(* Logix 5000 project; controller p65 vendor 1 type 14 code 85 rev 20.11; software revision 20.01; part 4 of 7 *)
(* tags used below, declared in another part *)
   DCMicroGridisInOperation : ALIAS FOR DINT00_23.8;
   DCMicroGridisSimulating : ALIAS FOR DINT00_23.10;
   House02accountBalance : ALIAS FOR REAL00_128;
   House02accountDepositRate : ALIAS FOR REAL00_129;
   House02Bclose : ALIAS FOR Local:3:O.Data.1;
   House02BcloseHILS : ALIAS FOR plc1_local_6[0].1;
   House02BcloseProxy : ALIAS FOR DINT00_28.31;
   House02BintReqClose : ALIAS FOR DINT00_29.0;
   House02BisClosed : ALIAS FOR DINT00_29.1;
   House02BisOpen : ALIAS FOR DINT00_29.2;
   House02BreqClose : ALIAS FOR DINT00_29.3;
   House02BreqOpen : ALIAS FOR DINT00_29.4;
   House02commandChanged : ALIAS FOR DINT00_29.5;
   House02commandChangedTimer : ALIAS FOR CLTIMER00_57;
   House02current : ALIAS FOR REAL00_130;
   House02currentHILS : ALIAS FOR plc1_local_2[1];
   House02currentRaw : ALIAS FOR Local:1:I.Ch13Data;
   House02deadband : ALIAS FOR REAL00_131;
   House02depositTimer : ALIAS FOR CLTIMER00_58;
   House02DisconnectPowerEventFail : ALIAS FOR DINT00_29.6;
   House02DisconnectPowerEventSuccess : ALIAS FOR DINT00_29.7;
   House02DisconnectPowerFailTimer : ALIAS FOR CLTIMER00_59;
   House02DisconnectPowerInProcess : ALIAS FOR DINT00_29.8;
   House02DisconnectPowerMsg : ALIAS FOR MESSAGE00_14;
   House02DisconnectPowerSuccessTimer : ALIAS FOR CLTIMER00_60;
   House02failedToConnect : ALIAS FOR DINT00_29.9;
   House02failedToDisconnect : ALIAS FOR DINT00_29.10;
   House02fundsAvailable : ALIAS FOR DINT00_29.11;
   House02incrementToAdd : ALIAS FOR REAL00_132;
   House02incrementToSubtract : ALIAS FOR REAL00_133;
   House02intReqConnect : ALIAS FOR DINT00_29.12;
   House02isConnected : ALIAS FOR DINT00_29.13;
   House02isDisconnected : ALIAS FOR DINT00_29.14;
   House02minBalance : ALIAS FOR REAL00_135;
   House02minBalanceToReconnect : ALIAS FOR REAL00_136;
   House02minTime : ALIAS FOR REAL00_137;
   House02powerRate : ALIAS FOR REAL00_138;
   House02powerRateMax : REAL;
   House02PurchasePowerEventFail : ALIAS FOR DINT00_29.15;
   House02PurchasePowerEventSuccess : ALIAS FOR DINT00_29.16;
   House02PurchasePowerFailTimer : ALIAS FOR CLTIMER00_61;
   House02PurchasePowerInProcess : ALIAS FOR DINT00_29.17;
   House02PurchasePowerMsg : ALIAS FOR MESSAGE00_15;
   House02PurchasePowerSuccessTimer : ALIAS FOR CLTIMER00_62;
   House02reqConnect : ALIAS FOR DINT00_29.18;
   House02reqDisconnect : ALIAS FOR DINT00_29.19;
   House02runningOut : ALIAS FOR DINT00_29.20;
   House02spendingRate : ALIAS FOR REAL00_139;
   House02timeRemaining : ALIAS FOR REAL00_140;
   House02usageTimer : ALIAS FOR CLTIMER00_63;
   House03accountBalance : ALIAS FOR REAL00_141;
   House03accountDepositRate : ALIAS FOR REAL00_142;
   House03Bclose : ALIAS FOR Local:3:O.Data.2;
   House03BcloseHILS : ALIAS FOR plc1_local_6[0].2;
   House03BcloseProxy : ALIAS FOR DINT00_29.21;
   House03BintReqClose : ALIAS FOR DINT00_29.22;
   House03BisClosed : ALIAS FOR DINT00_29.23;
   House03BisOpen : ALIAS FOR DINT00_29.24;
   House03BreqClose : ALIAS FOR DINT00_29.25;
   House03BreqOpen : ALIAS FOR DINT00_29.26;
   House03commandChanged : ALIAS FOR DINT00_29.27;
   House03commandChangedTimer : ALIAS FOR CLTIMER00_64;
   House03current : ALIAS FOR REAL00_143;
   House03currentHILS : ALIAS FOR plc1_local_2[2];
   House03currentRaw : ALIAS FOR Local:1:I.Ch14Data;
   House03deadband : ALIAS FOR REAL00_144;
   House03depositTimer : ALIAS FOR CLTIMER00_65;
   House03DisconnectPowerEventFail : ALIAS FOR DINT00_29.28;
   House03DisconnectPowerEventSuccess : ALIAS FOR DINT00_29.29;
   House03DisconnectPowerFailTimer : ALIAS FOR CLTIMER00_66;
   House03DisconnectPowerInProcess : ALIAS FOR DINT00_29.30;
   House03DisconnectPowerMsg : ALIAS FOR MESSAGE00_16;
   House03DisconnectPowerSuccessTimer : ALIAS FOR CLTIMER00_67;
   House03failedToConnect : ALIAS FOR DINT00_29.31;
   House03failedToDisconnect : ALIAS FOR DINT00_30.0;
   House03fundsAvailable : ALIAS FOR DINT00_30.1;
   House03incrementToAdd : ALIAS FOR REAL00_145;
   House03incrementToSubtract : ALIAS FOR REAL00_146;
   House03intReqConnect : ALIAS FOR DINT00_30.2;
   House03isConnected : ALIAS FOR DINT00_30.3;
   House03isDisconnected : ALIAS FOR DINT00_30.4;
   House03minBalance : ALIAS FOR REAL00_148;
   House03minBalanceToReconnect : ALIAS FOR REAL00_149;
   House03minTime : ALIAS FOR REAL00_150;
   House03powerRate : ALIAS FOR REAL00_151;
   House03powerRateMax : REAL;
   House03PurchasePowerEventFail : ALIAS FOR DINT00_30.5;
   House03PurchasePowerEventSuccess : ALIAS FOR DINT00_30.6;
   House03PurchasePowerFailTimer : ALIAS FOR CLTIMER00_68;
   House03PurchasePowerInProcess : ALIAS FOR DINT00_30.7;
   House03PurchasePowerMsg : ALIAS FOR MESSAGE00_17;
   House03PurchasePowerSuccessTimer : ALIAS FOR CLTIMER00_69;
   House03reqConnect : ALIAS FOR DINT00_30.8;
   House03reqDisconnect : ALIAS FOR DINT00_30.9;
   House03runningOut : ALIAS FOR DINT00_30.10;
   House03spendingRate : ALIAS FOR REAL00_152;
   House03timeRemaining : ALIAS FOR REAL00_153;
   House03usageTimer : ALIAS FOR CLTIMER00_70;
   House04accountBalance : ALIAS FOR REAL00_154;
   House04accountDepositRate : ALIAS FOR REAL00_155;
   House04Bclose : ALIAS FOR Local:3:O.Data.3;
   House04BcloseHILS : ALIAS FOR plc1_local_6[0].3;
   House04BcloseProxy : ALIAS FOR DINT00_30.11;
   House04BintReqClose : ALIAS FOR DINT00_30.12;
   House04BisClosed : ALIAS FOR DINT00_30.13;
   House04BisOpen : ALIAS FOR DINT00_30.14;
   House04BreqClose : ALIAS FOR DINT00_30.15;
   House04BreqOpen : ALIAS FOR DINT00_30.16;
   House04commandChanged : ALIAS FOR DINT00_30.17;
   House04commandChangedTimer : ALIAS FOR CLTIMER00_71;
   House04current : ALIAS FOR REAL00_156;
   House04currentHILS : ALIAS FOR plc1_local_2[3];
   House04currentRaw : ALIAS FOR Local:1:I.Ch15Data;
   House04deadband : ALIAS FOR REAL00_157;
   House04depositTimer : ALIAS FOR CLTIMER00_72;
   House04DisconnectPowerEventFail : ALIAS FOR DINT00_30.18;
   House04DisconnectPowerEventSuccess : ALIAS FOR DINT00_30.19;
   House04DisconnectPowerFailTimer : ALIAS FOR CLTIMER00_73;
   House04DisconnectPowerInProcess : ALIAS FOR DINT00_30.20;
   House04DisconnectPowerMsg : ALIAS FOR MESSAGE00_18;
   House04DisconnectPowerSuccessTimer : ALIAS FOR CLTIMER00_74;
   House04failedToConnect : ALIAS FOR DINT00_30.21;
   House04failedToDisconnect : ALIAS FOR DINT00_30.22;
   House04fundsAvailable : ALIAS FOR DINT00_30.23;
   House04incrementToAdd : ALIAS FOR REAL00_158;
   House04incrementToSubtract : ALIAS FOR REAL00_159;
   House04intReqConnect : ALIAS FOR DINT00_30.24;
   House04isConnected : ALIAS FOR DINT00_30.25;
   House04isDisconnected : ALIAS FOR DINT00_30.26;
   House04minBalance : ALIAS FOR REAL00_161;
   House04minBalanceToReconnect : ALIAS FOR REAL00_162;
   House04minTime : ALIAS FOR REAL00_163;
   House04powerRate : ALIAS FOR REAL00_164;
   House04powerRateMax : REAL;
   House04PurchasePowerEventFail : ALIAS FOR DINT00_30.27;
   House04PurchasePowerEventSuccess : ALIAS FOR DINT00_30.28;
   House04PurchasePowerFailTimer : ALIAS FOR CLTIMER00_75;
   House04PurchasePowerInProcess : ALIAS FOR DINT00_30.29;
   House04PurchasePowerMsg : ALIAS FOR MESSAGE00_19;
   House04PurchasePowerSuccessTimer : ALIAS FOR CLTIMER00_76;
   House04reqConnect : ALIAS FOR DINT00_30.30;
   House04reqDisconnect : ALIAS FOR DINT00_30.31;
   House04runningOut : ALIAS FOR DINT00_31.0;
   House04spendingRate : ALIAS FOR REAL00_165;
   House04timeRemaining : ALIAS FOR REAL00_166;
   House04usageTimer : ALIAS FOR CLTIMER00_77;
   LoadslowVoltage : ALIAS FOR DINT00_27.23;
   UsingAgents : BOOL;

PROGRAM House02   (* main routine House02 *)

ROUTINE House02   (* ladder *)
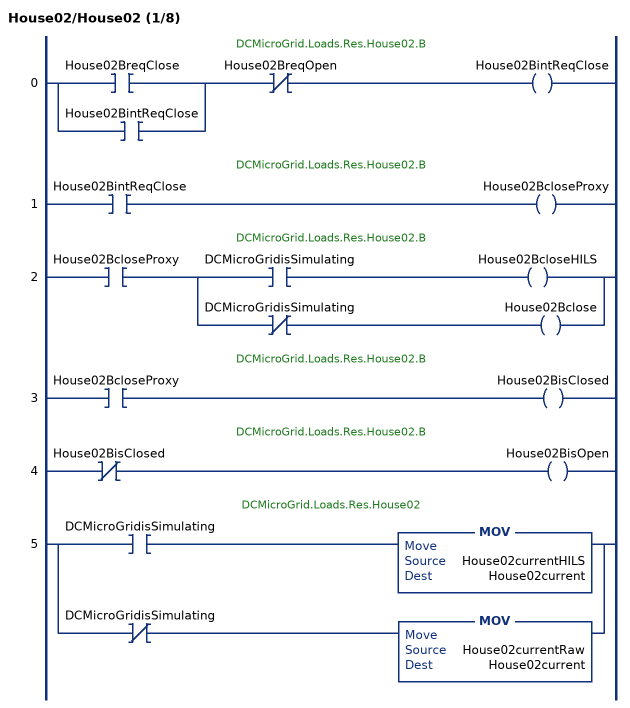
   // DCMicroGrid.Loads.Res.House02.B
   0: [XIC(House02BreqClose) ,XIC(House02BintReqClose) ]XIO(House02BreqOpen)OTE(House02BintReqClose);
   // DCMicroGrid.Loads.Res.House02.B
   1: XIC(House02BintReqClose)OTE(House02BcloseProxy);
   // DCMicroGrid.Loads.Res.House02.B
   2: XIC(House02BcloseProxy)[XIC(DCMicroGridisSimulating) OTE(House02BcloseHILS) ,XIO(DCMicroGridisSimulating) OTE(House02Bclose) ];
   // DCMicroGrid.Loads.Res.House02.B
   3: XIC(House02BcloseProxy)OTE(House02BisClosed);
   // DCMicroGrid.Loads.Res.House02.B
   4: XIO(House02BisClosed)OTE(House02BisOpen);
   // DCMicroGrid.Loads.Res.House02
   5: [XIC(DCMicroGridisSimulating) MOV(House02currentHILS,House02current) ,XIO(DCMicroGridisSimulating) MOV(House02currentRaw,House02current) ];
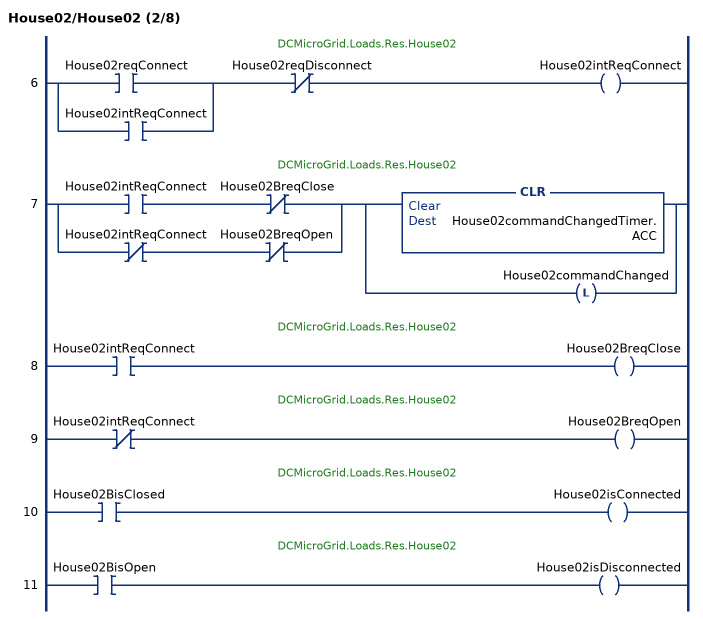
   // DCMicroGrid.Loads.Res.House02
   6: [XIC(House02reqConnect) ,XIC(House02intReqConnect) ]XIO(House02reqDisconnect)OTE(House02intReqConnect);
   // DCMicroGrid.Loads.Res.House02
   7: [XIC(House02intReqConnect) XIO(House02BreqClose) ,XIO(House02intReqConnect) XIO(House02BreqOpen) ][CLR(House02commandChangedTimer.ACC) ,OTL(House02commandChanged) ];
   // DCMicroGrid.Loads.Res.House02
   8: XIC(House02intReqConnect)OTE(House02BreqClose);
   // DCMicroGrid.Loads.Res.House02
   9: XIO(House02intReqConnect)OTE(House02BreqOpen);
   // DCMicroGrid.Loads.Res.House02
   10: XIC(House02BisClosed)OTE(House02isConnected);
   // DCMicroGrid.Loads.Res.House02
   11: XIC(House02BisOpen)OTE(House02isDisconnected);
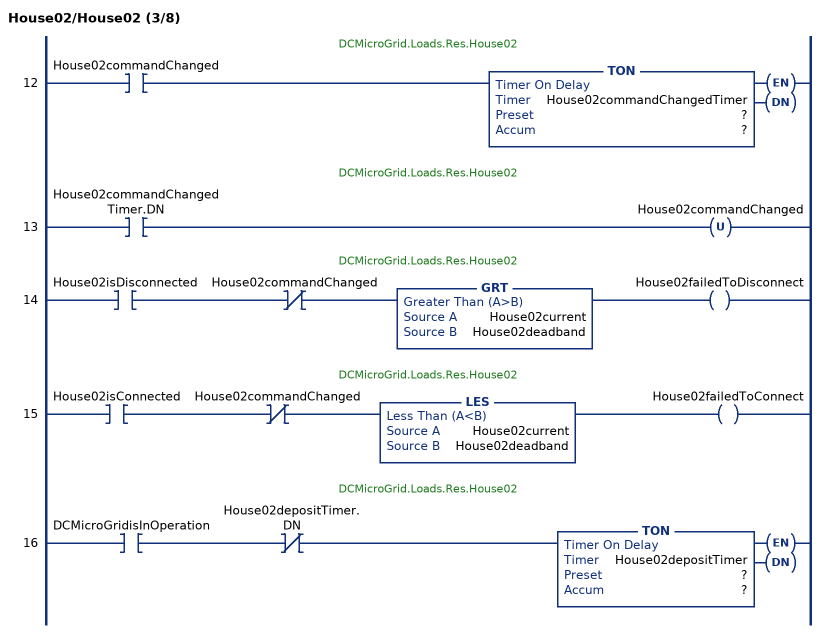
   // DCMicroGrid.Loads.Res.House02
   12: XIC(House02commandChanged)TON(House02commandChangedTimer,?,?);
   // DCMicroGrid.Loads.Res.House02
   13: XIC(House02commandChangedTimer.DN)OTU(House02commandChanged);
   // DCMicroGrid.Loads.Res.House02
   14: XIC(House02isDisconnected)XIO(House02commandChanged)GRT(House02current,House02deadband)OTE(House02failedToDisconnect);
   // DCMicroGrid.Loads.Res.House02
   15: XIC(House02isConnected)XIO(House02commandChanged)LES(House02current,House02deadband)OTE(House02failedToConnect);
   // DCMicroGrid.Loads.Res.House02
   16: XIC(DCMicroGridisInOperation)XIO(House02depositTimer.DN)TON(House02depositTimer,?,?);
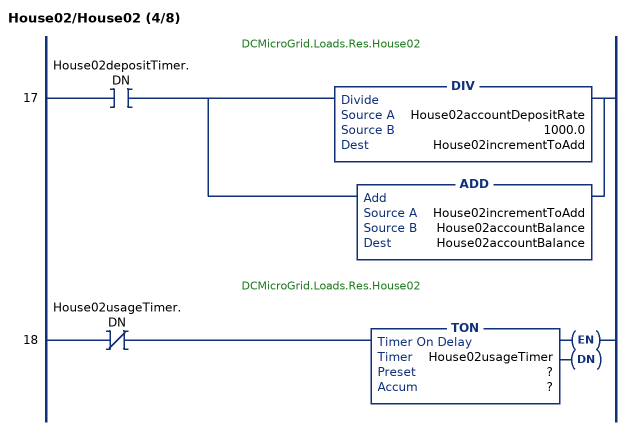
   // DCMicroGrid.Loads.Res.House02
   17: XIC(House02depositTimer.DN)[DIV(House02accountDepositRate,1000.0,House02incrementToAdd) ,ADD(House02incrementToAdd,House02accountBalance,House02accountBalance) ];
   // DCMicroGrid.Loads.Res.House02
   18: XIO(House02usageTimer.DN)TON(House02usageTimer,?,?);
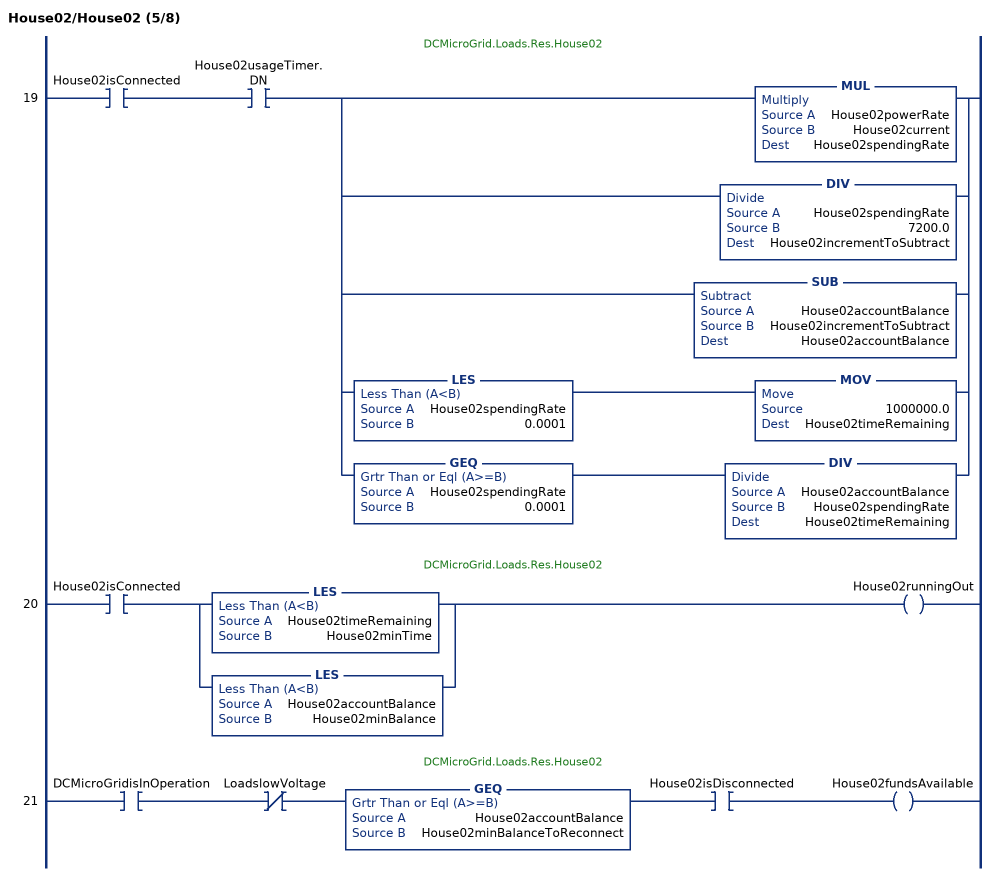
   // DCMicroGrid.Loads.Res.House02
   19: XIC(House02isConnected)XIC(House02usageTimer.DN)[MUL(House02powerRate,House02current,House02spendingRate) ,DIV(House02spendingRate,7200.0,House02incrementToSubtract) ,SUB(House02accountBalance,House02incrementToSubtract,House02accountBalance) ,[LES(House02spendingRate,0.0001) MOV(1000000.0,House02timeRemaining) ,GEQ(House02spendingRate,0.0001) DIV(House02accountBalance,House02spendingRate,House02timeRemaining) ] ];
   // DCMicroGrid.Loads.Res.House02
   20: XIC(House02isConnected)[LES(House02timeRemaining,House02minTime) ,LES(House02accountBalance,House02minBalance) ]OTE(House02runningOut);
   // DCMicroGrid.Loads.Res.House02
   21: XIC(DCMicroGridisInOperation)XIO(LoadslowVoltage)GEQ(House02accountBalance,House02minBalanceToReconnect)XIC(House02isDisconnected)OTE(House02fundsAvailable);
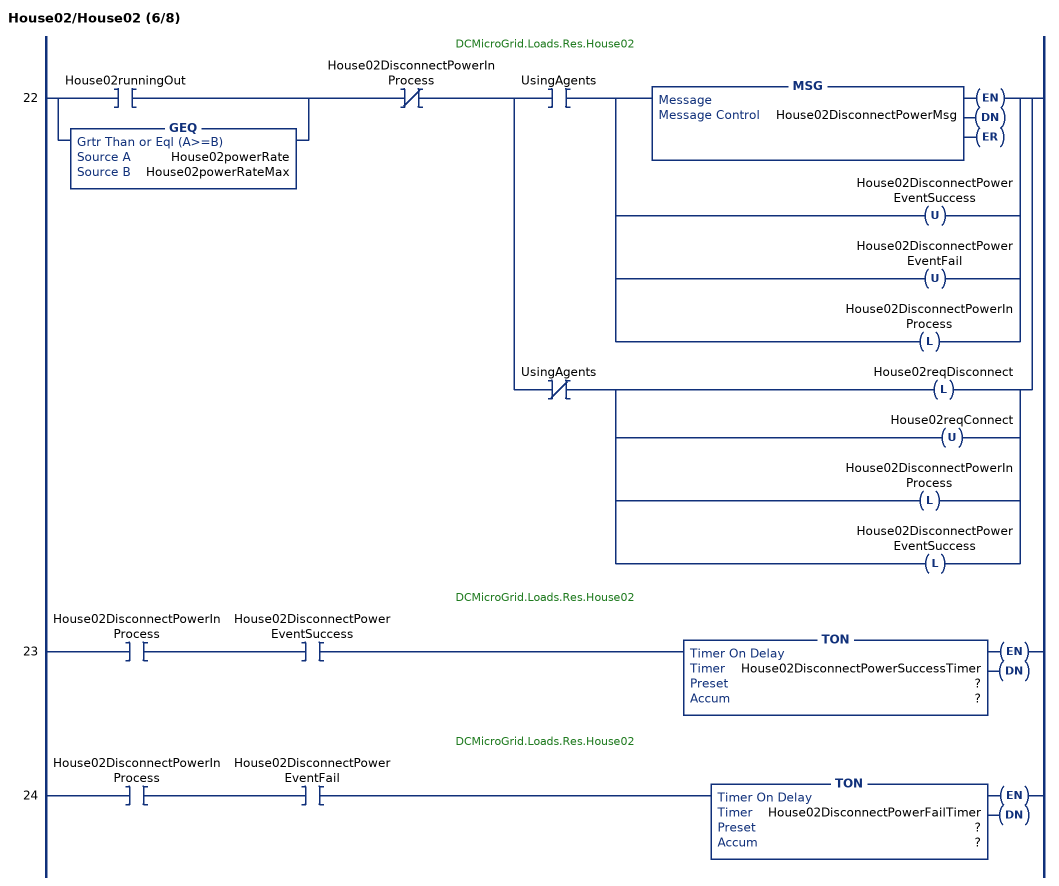
   // DCMicroGrid.Loads.Res.House02
   22: [XIC(House02runningOut) ,GEQ(House02powerRate,House02powerRateMax) ]XIO(House02DisconnectPowerInProcess)[XIC(UsingAgents) [MSG(House02DisconnectPowerMsg) ,OTU(House02DisconnectPowerEventSuccess) ,OTU(House02DisconnectPowerEventFail) ,OTL(House02DisconnectPowerInProcess) ] ,XIO(UsingAgents) [OTL(House02reqDisconnect) ,OTU(House02reqConnect) ,OTL(House02DisconnectPowerInProcess) ,OTL(House02DisconnectPowerEventSuccess) ] ];
   // DCMicroGrid.Loads.Res.House02
   23: XIC(House02DisconnectPowerInProcess)XIC(House02DisconnectPowerEventSuccess)TON(House02DisconnectPowerSuccessTimer,?,?);
   // DCMicroGrid.Loads.Res.House02
   24: XIC(House02DisconnectPowerInProcess)XIC(House02DisconnectPowerEventFail)TON(House02DisconnectPowerFailTimer,?,?);
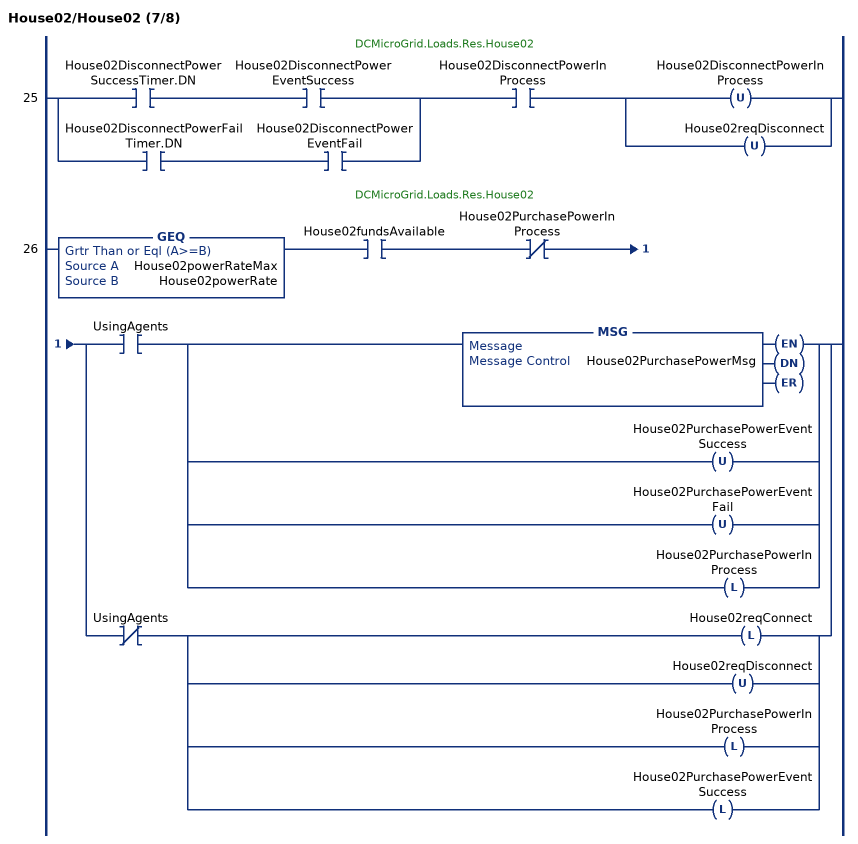
   // DCMicroGrid.Loads.Res.House02
   25: [XIC(House02DisconnectPowerSuccessTimer.DN) XIC(House02DisconnectPowerEventSuccess) ,XIC(House02DisconnectPowerFailTimer.DN) XIC(House02DisconnectPowerEventFail) ]XIC(House02DisconnectPowerInProcess)[OTU(House02DisconnectPowerInProcess) ,OTU(House02reqDisconnect) ];
   // DCMicroGrid.Loads.Res.House02
   26: GEQ(House02powerRateMax,House02powerRate)XIC(House02fundsAvailable)XIO(House02PurchasePowerInProcess)[XIC(UsingAgents) [MSG(House02PurchasePowerMsg) ,OTU(House02PurchasePowerEventSuccess) ,OTU(House02PurchasePowerEventFail) ,OTL(House02PurchasePowerInProcess) ] ,XIO(UsingAgents) [OTL(House02reqConnect) ,OTU(House02reqDisconnect) ,OTL(House02PurchasePowerInProcess) ,OTL(House02PurchasePowerEventSuccess) ] ];
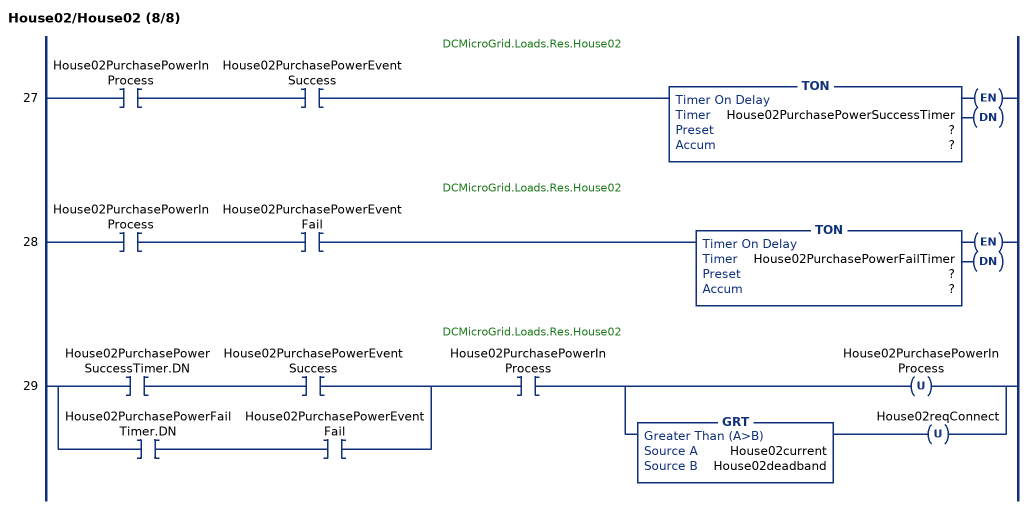
   // DCMicroGrid.Loads.Res.House02
   27: XIC(House02PurchasePowerInProcess)XIC(House02PurchasePowerEventSuccess)TON(House02PurchasePowerSuccessTimer,?,?);
   // DCMicroGrid.Loads.Res.House02
   28: XIC(House02PurchasePowerInProcess)XIC(House02PurchasePowerEventFail)TON(House02PurchasePowerFailTimer,?,?);
   // DCMicroGrid.Loads.Res.House02
   29: [XIC(House02PurchasePowerSuccessTimer.DN) XIC(House02PurchasePowerEventSuccess) ,XIC(House02PurchasePowerFailTimer.DN) XIC(House02PurchasePowerEventFail) ]XIC(House02PurchasePowerInProcess)[OTU(House02PurchasePowerInProcess) ,GRT(House02current,House02deadband) OTU(House02reqConnect) ];
END_ROUTINE
END_PROGRAM

PROGRAM House03   (* main routine House03 *)

ROUTINE House03   (* ladder *)
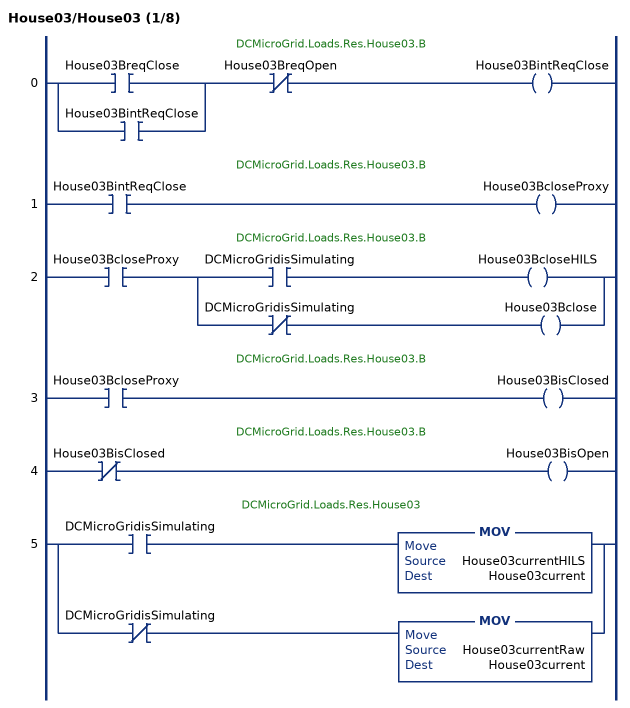
   // DCMicroGrid.Loads.Res.House03.B
   0: [XIC(House03BreqClose) ,XIC(House03BintReqClose) ]XIO(House03BreqOpen)OTE(House03BintReqClose);
   // DCMicroGrid.Loads.Res.House03.B
   1: XIC(House03BintReqClose)OTE(House03BcloseProxy);
   // DCMicroGrid.Loads.Res.House03.B
   2: XIC(House03BcloseProxy)[XIC(DCMicroGridisSimulating) OTE(House03BcloseHILS) ,XIO(DCMicroGridisSimulating) OTE(House03Bclose) ];
   // DCMicroGrid.Loads.Res.House03.B
   3: XIC(House03BcloseProxy)OTE(House03BisClosed);
   // DCMicroGrid.Loads.Res.House03.B
   4: XIO(House03BisClosed)OTE(House03BisOpen);
   // DCMicroGrid.Loads.Res.House03
   5: [XIC(DCMicroGridisSimulating) MOV(House03currentHILS,House03current) ,XIO(DCMicroGridisSimulating) MOV(House03currentRaw,House03current) ];
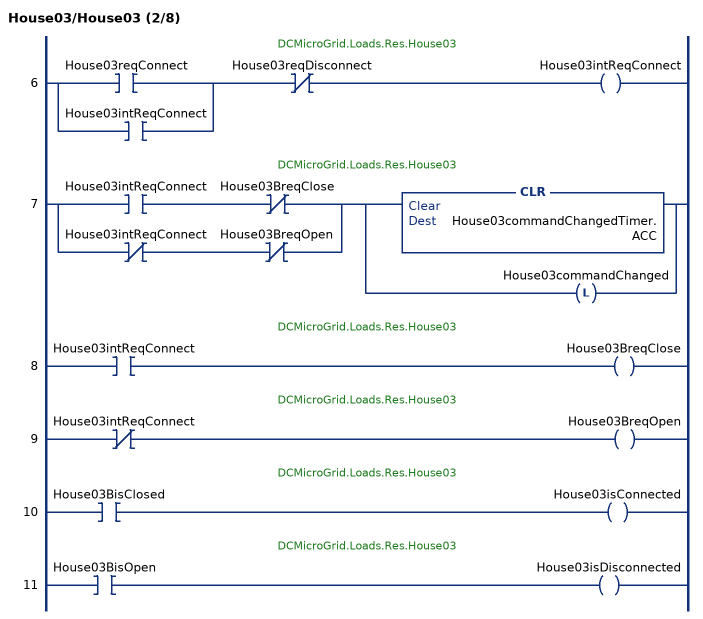
   // DCMicroGrid.Loads.Res.House03
   6: [XIC(House03reqConnect) ,XIC(House03intReqConnect) ]XIO(House03reqDisconnect)OTE(House03intReqConnect);
   // DCMicroGrid.Loads.Res.House03
   7: [XIC(House03intReqConnect) XIO(House03BreqClose) ,XIO(House03intReqConnect) XIO(House03BreqOpen) ][CLR(House03commandChangedTimer.ACC) ,OTL(House03commandChanged) ];
   // DCMicroGrid.Loads.Res.House03
   8: XIC(House03intReqConnect)OTE(House03BreqClose);
   // DCMicroGrid.Loads.Res.House03
   9: XIO(House03intReqConnect)OTE(House03BreqOpen);
   // DCMicroGrid.Loads.Res.House03
   10: XIC(House03BisClosed)OTE(House03isConnected);
   // DCMicroGrid.Loads.Res.House03
   11: XIC(House03BisOpen)OTE(House03isDisconnected);
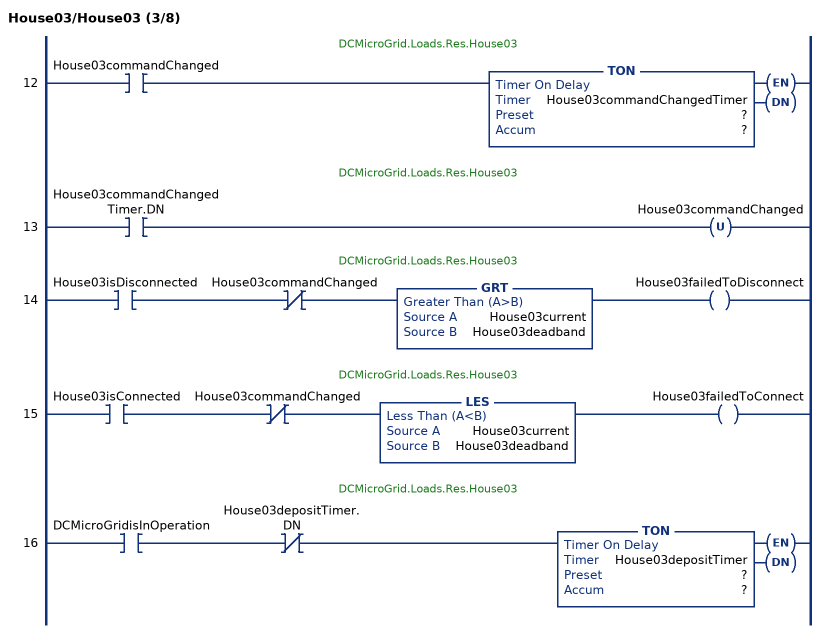
   // DCMicroGrid.Loads.Res.House03
   12: XIC(House03commandChanged)TON(House03commandChangedTimer,?,?);
   // DCMicroGrid.Loads.Res.House03
   13: XIC(House03commandChangedTimer.DN)OTU(House03commandChanged);
   // DCMicroGrid.Loads.Res.House03
   14: XIC(House03isDisconnected)XIO(House03commandChanged)GRT(House03current,House03deadband)OTE(House03failedToDisconnect);
   // DCMicroGrid.Loads.Res.House03
   15: XIC(House03isConnected)XIO(House03commandChanged)LES(House03current,House03deadband)OTE(House03failedToConnect);
   // DCMicroGrid.Loads.Res.House03
   16: XIC(DCMicroGridisInOperation)XIO(House03depositTimer.DN)TON(House03depositTimer,?,?);
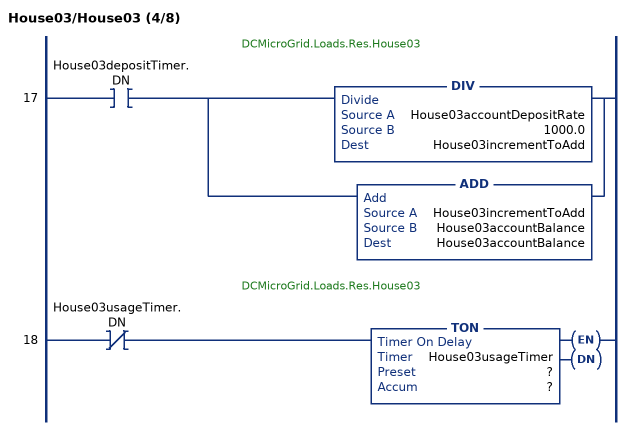
   // DCMicroGrid.Loads.Res.House03
   17: XIC(House03depositTimer.DN)[DIV(House03accountDepositRate,1000.0,House03incrementToAdd) ,ADD(House03incrementToAdd,House03accountBalance,House03accountBalance) ];
   // DCMicroGrid.Loads.Res.House03
   18: XIO(House03usageTimer.DN)TON(House03usageTimer,?,?);
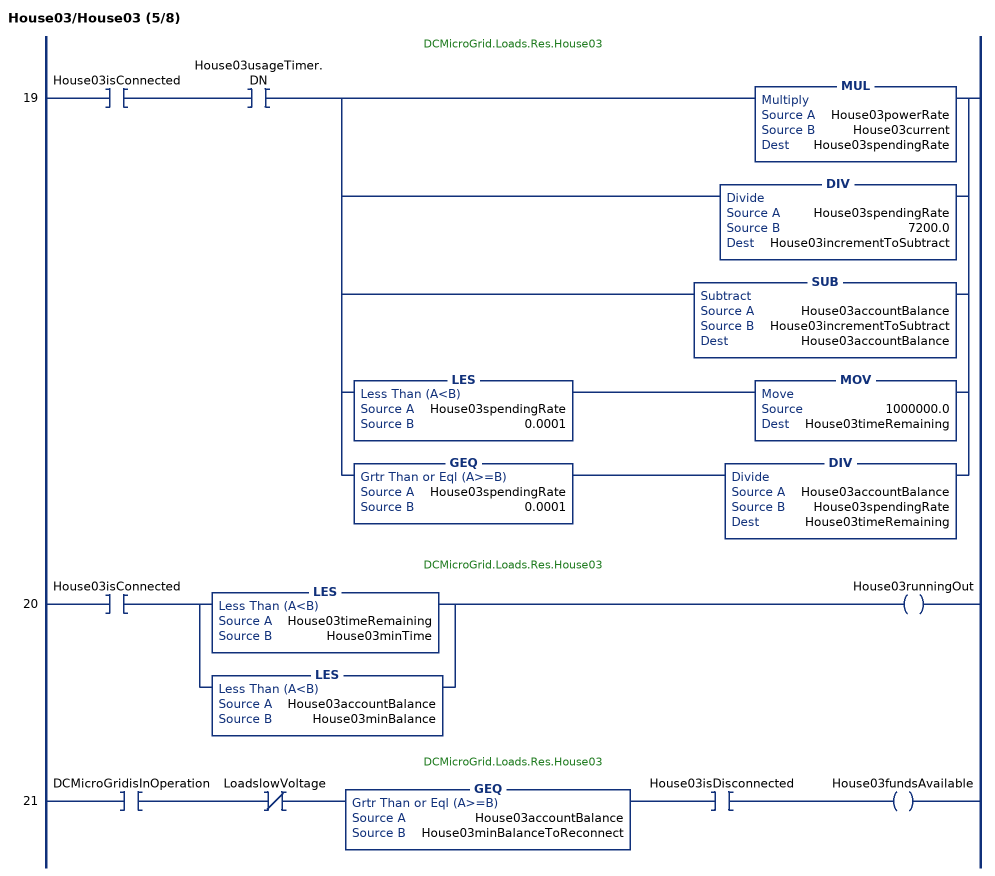
   // DCMicroGrid.Loads.Res.House03
   19: XIC(House03isConnected)XIC(House03usageTimer.DN)[MUL(House03powerRate,House03current,House03spendingRate) ,DIV(House03spendingRate,7200.0,House03incrementToSubtract) ,SUB(House03accountBalance,House03incrementToSubtract,House03accountBalance) ,[LES(House03spendingRate,0.0001) MOV(1000000.0,House03timeRemaining) ,GEQ(House03spendingRate,0.0001) DIV(House03accountBalance,House03spendingRate,House03timeRemaining) ] ];
   // DCMicroGrid.Loads.Res.House03
   20: XIC(House03isConnected)[LES(House03timeRemaining,House03minTime) ,LES(House03accountBalance,House03minBalance) ]OTE(House03runningOut);
   // DCMicroGrid.Loads.Res.House03
   21: XIC(DCMicroGridisInOperation)XIO(LoadslowVoltage)GEQ(House03accountBalance,House03minBalanceToReconnect)XIC(House03isDisconnected)OTE(House03fundsAvailable);
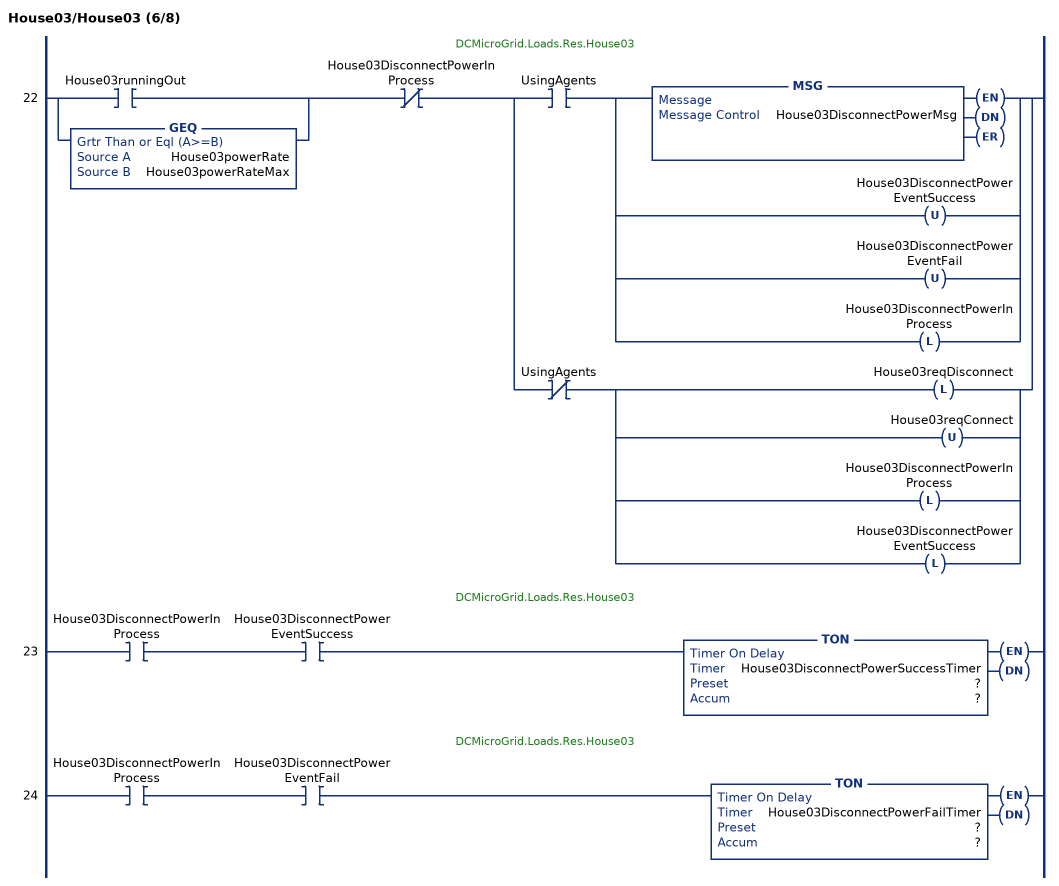
   // DCMicroGrid.Loads.Res.House03
   22: [XIC(House03runningOut) ,GEQ(House03powerRate,House03powerRateMax) ]XIO(House03DisconnectPowerInProcess)[XIC(UsingAgents) [MSG(House03DisconnectPowerMsg) ,OTU(House03DisconnectPowerEventSuccess) ,OTU(House03DisconnectPowerEventFail) ,OTL(House03DisconnectPowerInProcess) ] ,XIO(UsingAgents) [OTL(House03reqDisconnect) ,OTU(House03reqConnect) ,OTL(House03DisconnectPowerInProcess) ,OTL(House03DisconnectPowerEventSuccess) ] ];
   // DCMicroGrid.Loads.Res.House03
   23: XIC(House03DisconnectPowerInProcess)XIC(House03DisconnectPowerEventSuccess)TON(House03DisconnectPowerSuccessTimer,?,?);
   // DCMicroGrid.Loads.Res.House03
   24: XIC(House03DisconnectPowerInProcess)XIC(House03DisconnectPowerEventFail)TON(House03DisconnectPowerFailTimer,?,?);
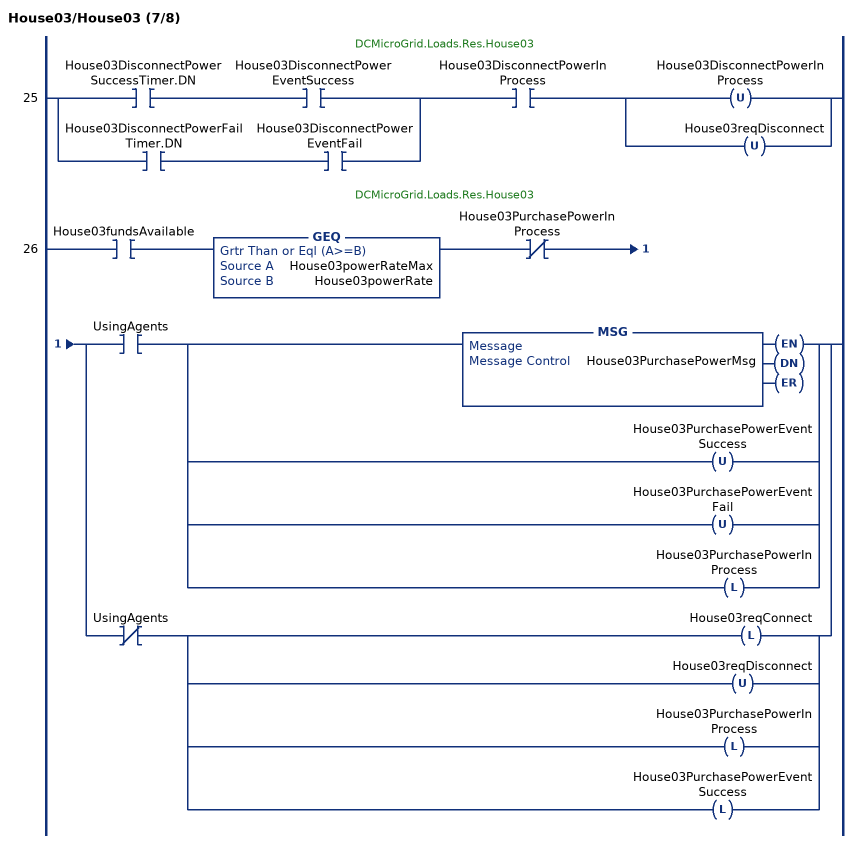
   // DCMicroGrid.Loads.Res.House03
   25: [XIC(House03DisconnectPowerSuccessTimer.DN) XIC(House03DisconnectPowerEventSuccess) ,XIC(House03DisconnectPowerFailTimer.DN) XIC(House03DisconnectPowerEventFail) ]XIC(House03DisconnectPowerInProcess)[OTU(House03DisconnectPowerInProcess) ,OTU(House03reqDisconnect) ];
   // DCMicroGrid.Loads.Res.House03
   26: XIC(House03fundsAvailable)GEQ(House03powerRateMax,House03powerRate)XIO(House03PurchasePowerInProcess)[XIC(UsingAgents) [MSG(House03PurchasePowerMsg) ,OTU(House03PurchasePowerEventSuccess) ,OTU(House03PurchasePowerEventFail) ,OTL(House03PurchasePowerInProcess) ] ,XIO(UsingAgents) [OTL(House03reqConnect) ,OTU(House03reqDisconnect) ,OTL(House03PurchasePowerInProcess) ,OTL(House03PurchasePowerEventSuccess) ] ];
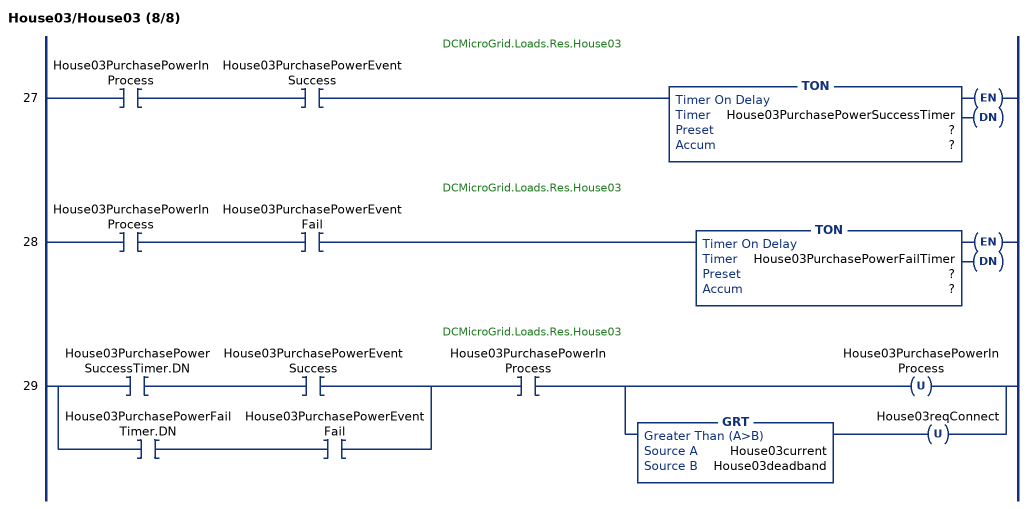
   // DCMicroGrid.Loads.Res.House03
   27: XIC(House03PurchasePowerInProcess)XIC(House03PurchasePowerEventSuccess)TON(House03PurchasePowerSuccessTimer,?,?);
   // DCMicroGrid.Loads.Res.House03
   28: XIC(House03PurchasePowerInProcess)XIC(House03PurchasePowerEventFail)TON(House03PurchasePowerFailTimer,?,?);
   // DCMicroGrid.Loads.Res.House03
   29: [XIC(House03PurchasePowerSuccessTimer.DN) XIC(House03PurchasePowerEventSuccess) ,XIC(House03PurchasePowerFailTimer.DN) XIC(House03PurchasePowerEventFail) ]XIC(House03PurchasePowerInProcess)[OTU(House03PurchasePowerInProcess) ,GRT(House03current,House03deadband) OTU(House03reqConnect) ];
END_ROUTINE
END_PROGRAM

PROGRAM House04   (* main routine House04 *)

ROUTINE House04   (* ladder *)
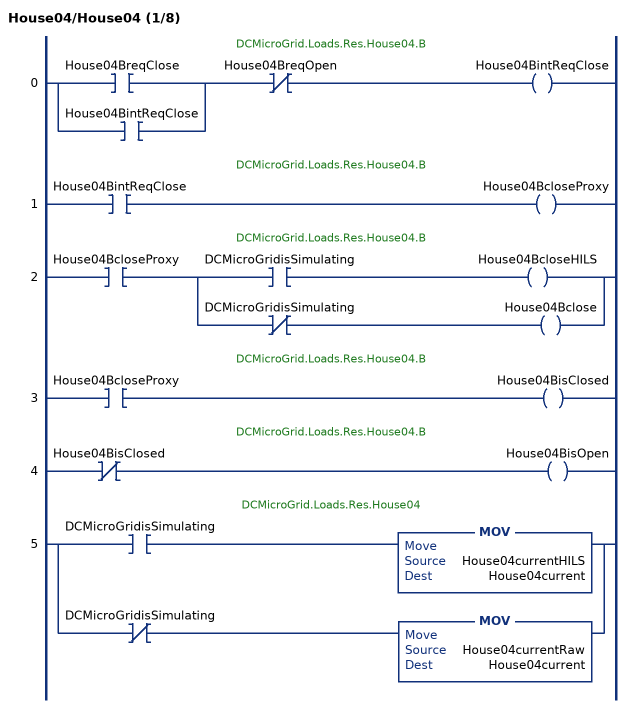
   // DCMicroGrid.Loads.Res.House04.B
   0: [XIC(House04BreqClose) ,XIC(House04BintReqClose) ]XIO(House04BreqOpen)OTE(House04BintReqClose);
   // DCMicroGrid.Loads.Res.House04.B
   1: XIC(House04BintReqClose)OTE(House04BcloseProxy);
   // DCMicroGrid.Loads.Res.House04.B
   2: XIC(House04BcloseProxy)[XIC(DCMicroGridisSimulating) OTE(House04BcloseHILS) ,XIO(DCMicroGridisSimulating) OTE(House04Bclose) ];
   // DCMicroGrid.Loads.Res.House04.B
   3: XIC(House04BcloseProxy)OTE(House04BisClosed);
   // DCMicroGrid.Loads.Res.House04.B
   4: XIO(House04BisClosed)OTE(House04BisOpen);
   // DCMicroGrid.Loads.Res.House04
   5: [XIC(DCMicroGridisSimulating) MOV(House04currentHILS,House04current) ,XIO(DCMicroGridisSimulating) MOV(House04currentRaw,House04current) ];
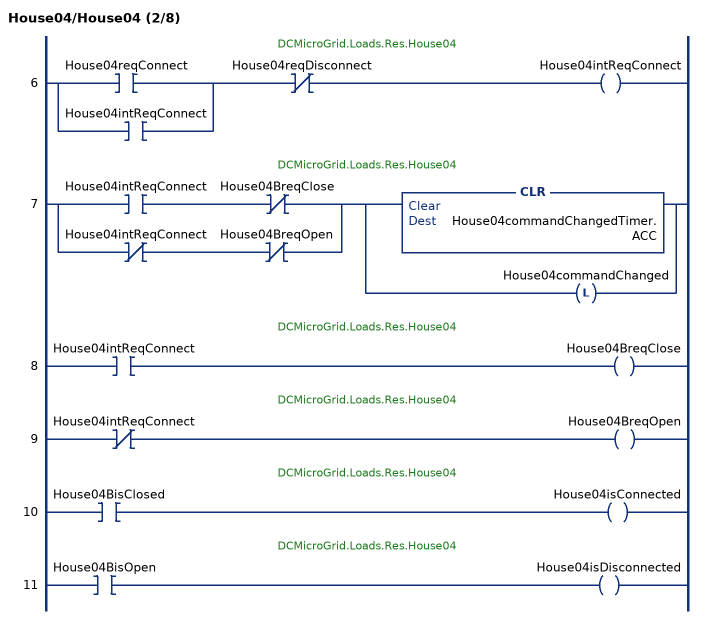
   // DCMicroGrid.Loads.Res.House04
   6: [XIC(House04reqConnect) ,XIC(House04intReqConnect) ]XIO(House04reqDisconnect)OTE(House04intReqConnect);
   // DCMicroGrid.Loads.Res.House04
   7: [XIC(House04intReqConnect) XIO(House04BreqClose) ,XIO(House04intReqConnect) XIO(House04BreqOpen) ][CLR(House04commandChangedTimer.ACC) ,OTL(House04commandChanged) ];
   // DCMicroGrid.Loads.Res.House04
   8: XIC(House04intReqConnect)OTE(House04BreqClose);
   // DCMicroGrid.Loads.Res.House04
   9: XIO(House04intReqConnect)OTE(House04BreqOpen);
   // DCMicroGrid.Loads.Res.House04
   10: XIC(House04BisClosed)OTE(House04isConnected);
   // DCMicroGrid.Loads.Res.House04
   11: XIC(House04BisOpen)OTE(House04isDisconnected);
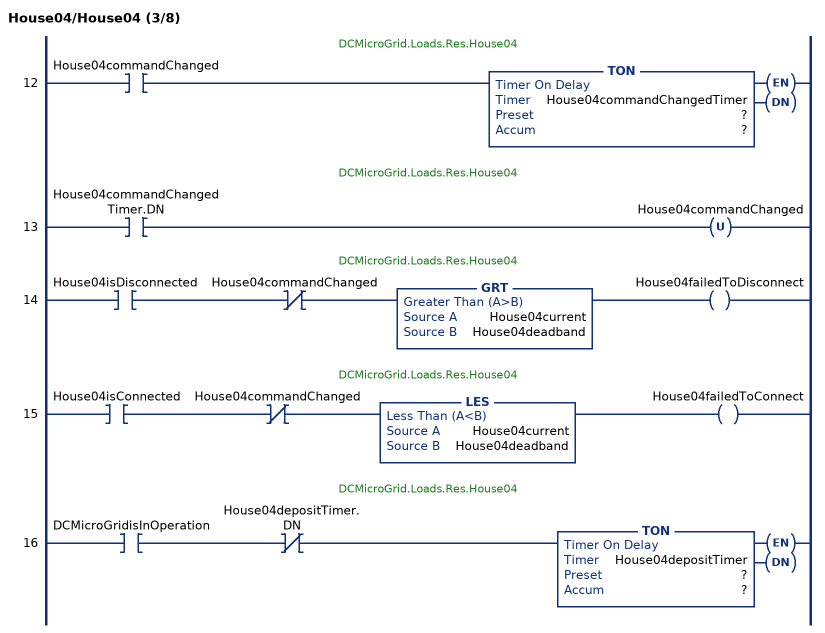
   // DCMicroGrid.Loads.Res.House04
   12: XIC(House04commandChanged)TON(House04commandChangedTimer,?,?);
   // DCMicroGrid.Loads.Res.House04
   13: XIC(House04commandChangedTimer.DN)OTU(House04commandChanged);
   // DCMicroGrid.Loads.Res.House04
   14: XIC(House04isDisconnected)XIO(House04commandChanged)GRT(House04current,House04deadband)OTE(House04failedToDisconnect);
   // DCMicroGrid.Loads.Res.House04
   15: XIC(House04isConnected)XIO(House04commandChanged)LES(House04current,House04deadband)OTE(House04failedToConnect);
   // DCMicroGrid.Loads.Res.House04
   16: XIC(DCMicroGridisInOperation)XIO(House04depositTimer.DN)TON(House04depositTimer,?,?);
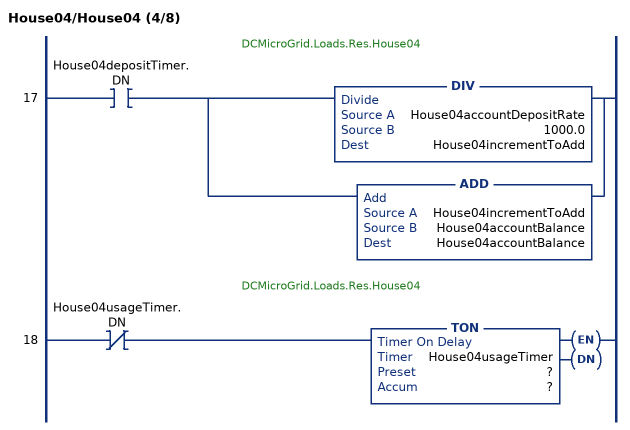
   // DCMicroGrid.Loads.Res.House04
   17: XIC(House04depositTimer.DN)[DIV(House04accountDepositRate,1000.0,House04incrementToAdd) ,ADD(House04incrementToAdd,House04accountBalance,House04accountBalance) ];
   // DCMicroGrid.Loads.Res.House04
   18: XIO(House04usageTimer.DN)TON(House04usageTimer,?,?);
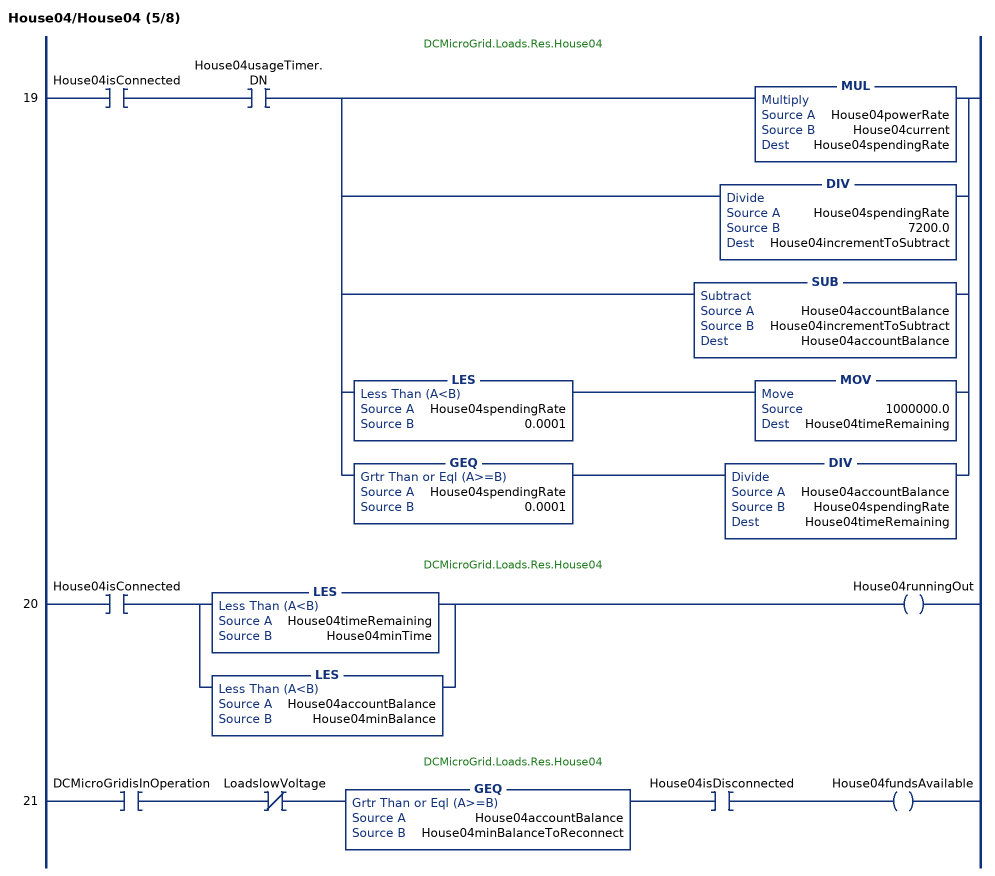
   // DCMicroGrid.Loads.Res.House04
   19: XIC(House04isConnected)XIC(House04usageTimer.DN)[MUL(House04powerRate,House04current,House04spendingRate) ,DIV(House04spendingRate,7200.0,House04incrementToSubtract) ,SUB(House04accountBalance,House04incrementToSubtract,House04accountBalance) ,[LES(House04spendingRate,0.0001) MOV(1000000.0,House04timeRemaining) ,GEQ(House04spendingRate,0.0001) DIV(House04accountBalance,House04spendingRate,House04timeRemaining) ] ];
   // DCMicroGrid.Loads.Res.House04
   20: XIC(House04isConnected)[LES(House04timeRemaining,House04minTime) ,LES(House04accountBalance,House04minBalance) ]OTE(House04runningOut);
   // DCMicroGrid.Loads.Res.House04
   21: XIC(DCMicroGridisInOperation)XIO(LoadslowVoltage)GEQ(House04accountBalance,House04minBalanceToReconnect)XIC(House04isDisconnected)OTE(House04fundsAvailable);
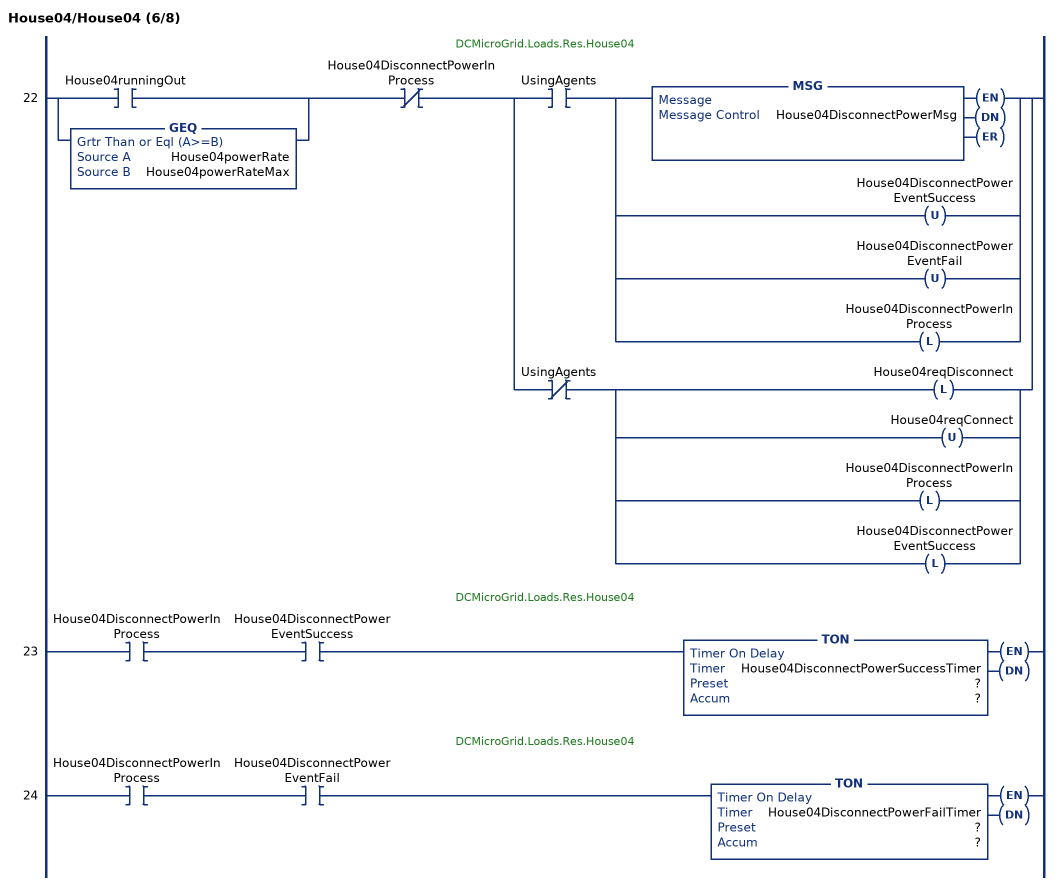
   // DCMicroGrid.Loads.Res.House04
   22: [XIC(House04runningOut) ,GEQ(House04powerRate,House04powerRateMax) ]XIO(House04DisconnectPowerInProcess)[XIC(UsingAgents) [MSG(House04DisconnectPowerMsg) ,OTU(House04DisconnectPowerEventSuccess) ,OTU(House04DisconnectPowerEventFail) ,OTL(House04DisconnectPowerInProcess) ] ,XIO(UsingAgents) [OTL(House04reqDisconnect) ,OTU(House04reqConnect) ,OTL(House04DisconnectPowerInProcess) ,OTL(House04DisconnectPowerEventSuccess) ] ];
   // DCMicroGrid.Loads.Res.House04
   23: XIC(House04DisconnectPowerInProcess)XIC(House04DisconnectPowerEventSuccess)TON(House04DisconnectPowerSuccessTimer,?,?);
   // DCMicroGrid.Loads.Res.House04
   24: XIC(House04DisconnectPowerInProcess)XIC(House04DisconnectPowerEventFail)TON(House04DisconnectPowerFailTimer,?,?);
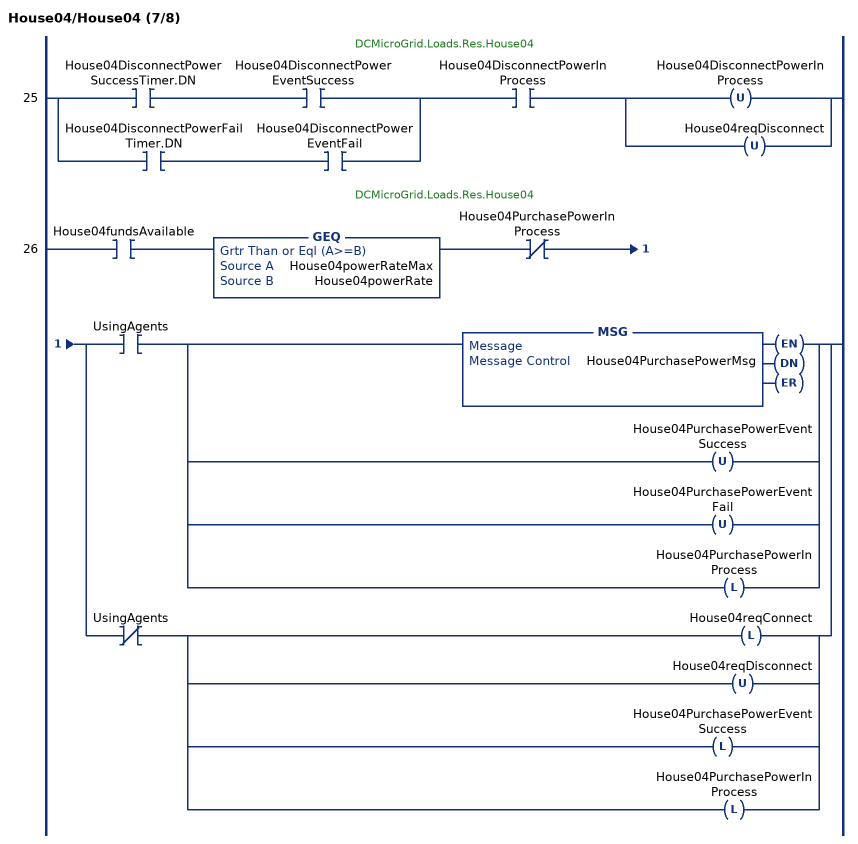
   // DCMicroGrid.Loads.Res.House04
   25: [XIC(House04DisconnectPowerSuccessTimer.DN) XIC(House04DisconnectPowerEventSuccess) ,XIC(House04DisconnectPowerFailTimer.DN) XIC(House04DisconnectPowerEventFail) ]XIC(House04DisconnectPowerInProcess)[OTU(House04DisconnectPowerInProcess) ,OTU(House04reqDisconnect) ];
   // DCMicroGrid.Loads.Res.House04
   26: XIC(House04fundsAvailable)GEQ(House04powerRateMax,House04powerRate)XIO(House04PurchasePowerInProcess)[XIC(UsingAgents) [MSG(House04PurchasePowerMsg) ,OTU(House04PurchasePowerEventSuccess) ,OTU(House04PurchasePowerEventFail) ,OTL(House04PurchasePowerInProcess) ] ,XIO(UsingAgents) [OTL(House04reqConnect) ,OTU(House04reqDisconnect) ,OTL(House04PurchasePowerEventSuccess) ,OTL(House04PurchasePowerInProcess) ] ];
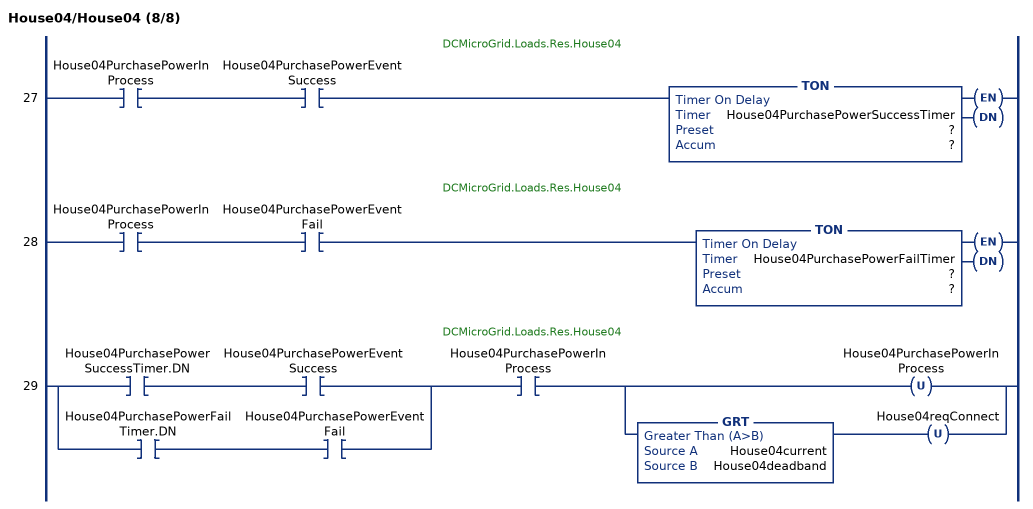
   // DCMicroGrid.Loads.Res.House04
   27: XIC(House04PurchasePowerInProcess)XIC(House04PurchasePowerEventSuccess)TON(House04PurchasePowerSuccessTimer,?,?);
   // DCMicroGrid.Loads.Res.House04
   28: XIC(House04PurchasePowerInProcess)XIC(House04PurchasePowerEventFail)TON(House04PurchasePowerFailTimer,?,?);
   // DCMicroGrid.Loads.Res.House04
   29: [XIC(House04PurchasePowerSuccessTimer.DN) XIC(House04PurchasePowerEventSuccess) ,XIC(House04PurchasePowerFailTimer.DN) XIC(House04PurchasePowerEventFail) ]XIC(House04PurchasePowerInProcess)[OTU(House04PurchasePowerInProcess) ,GRT(House04current,House04deadband) OTU(House04reqConnect) ];
END_ROUTINE
END_PROGRAM
